(* IEC 61131-3 sources: Elmo_Master/Lasal_PRG/Elmo_EtherCAT_Test_4Axis/Class/SimulationSetup, 1 file *)

(* ---- SimulationSetup.st ---- *)
(*!
<Class
	Name               = "SimulationSetup"
	Revision           = "0.0"
	RealtimeTask       = "false"
	CyclicTask         = "false"
	BackgroundTask     = "false"
	Sigmatek           = "false"
	OSInterface        = "false"
	HighPriority       = "false"
	Automatic          = "false"
	UpdateMode         = "Prescan"
	SharedCommandTable = "true"
	Objectsize         = "(422,120)">
	<Channels>
		<Server Name="Axis_1" Visualized="false" Initialize="true" WriteProtected="false" Retentive="File"/>
		<Server Name="Axis_2" Visualized="false" Initialize="true" WriteProtected="false" Retentive="File"/>
		<Server Name="Axis_3" Visualized="false" Initialize="true" WriteProtected="false" Retentive="File"/>
		<Server Name="Axis_4" Visualized="false" Initialize="true" WriteProtected="false" Retentive="File"/>
		<Server Name="Axis_5" Visualized="false" Initialize="true" WriteProtected="false" Retentive="File"/>
		<Server Name="Axis_6" Visualized="false" Initialize="true" WriteProtected="false" Retentive="File"/>
		<Server Name="Axis_7" Visualized="false" Initialize="true" WriteProtected="false" Retentive="File"/>
		<Server Name="Axis_8" Visualized="false" Initialize="true" WriteProtected="false" Retentive="File"/>
		<Server Name="Axis_9" Visualized="false" Initialize="true" WriteProtected="false" Retentive="File"/>
		<Server Name="ClassSvr" Visualized="false" Initialize="false" WriteProtected="true" Retentive="false"/>
		<Client Name="Simul_Axis_1" Required="false" Internal="false"/>
		<Client Name="Simul_Axis_2" Required="false" Internal="false"/>
		<Client Name="Simul_Axis_3" Required="false" Internal="false"/>
		<Client Name="Simul_Axis_4" Required="false" Internal="false"/>
		<Client Name="Simul_Axis_5" Required="false" Internal="false"/>
		<Client Name="Simul_Axis_6" Required="false" Internal="false"/>
		<Client Name="Simul_Axis_7" Required="false" Internal="false"/>
		<Client Name="Simul_Axis_8" Required="false" Internal="false"/>
		<Client Name="Simul_Axis_9" Required="false" Internal="false"/>
	</Channels>
</Class>
*)
SimulationSetup : CLASS
  //Servers:
	ClassSvr 	: SvrChCmd_DINT;
	Axis_1 	: SvrCh_DINT;
	Axis_2 	: SvrCh_DINT;
	Axis_3 	: SvrCh_DINT;
	Axis_4 	: SvrCh_DINT;
	Axis_5 	: SvrCh_DINT;
	Axis_6 	: SvrCh_DINT;
	Axis_7 	: SvrCh_DINT;
	Axis_8 	: SvrCh_DINT;
	Axis_9 	: SvrCh_DINT;
  //Clients:
	Simul_Axis_1 	: CltCh_DINT;
	Simul_Axis_2 	: CltCh_DINT;
	Simul_Axis_3 	: CltCh_DINT;
	Simul_Axis_4 	: CltCh_DINT;
	Simul_Axis_5 	: CltCh_DINT;
	Simul_Axis_6 	: CltCh_DINT;
	Simul_Axis_7 	: CltCh_DINT;
	Simul_Axis_8 	: CltCh_DINT;
	Simul_Axis_9 	: CltCh_DINT;
  //Variables:
  //Functions:

	FUNCTION VIRTUAL GLOBAL Init;

	FUNCTION Write_Simul
		VAR_INPUT
			Index 	: DINT;
			Value 	: DINT;
		END_VAR;

	FUNCTION VIRTUAL GLOBAL Axis_1::Write
		VAR_INPUT
			input (EAX) 	: DINT;
		END_VAR
		VAR_OUTPUT
			result (EAX) 	: DINT;
		END_VAR;

	FUNCTION VIRTUAL GLOBAL Axis_2::Write
		VAR_INPUT
			input (EAX) 	: DINT;
		END_VAR
		VAR_OUTPUT
			result (EAX) 	: DINT;
		END_VAR;

	FUNCTION VIRTUAL GLOBAL Axis_3::Write
		VAR_INPUT
			input (EAX) 	: DINT;
		END_VAR
		VAR_OUTPUT
			result (EAX) 	: DINT;
		END_VAR;

	FUNCTION VIRTUAL GLOBAL Axis_4::Write
		VAR_INPUT
			input (EAX) 	: DINT;
		END_VAR
		VAR_OUTPUT
			result (EAX) 	: DINT;
		END_VAR;

	FUNCTION VIRTUAL GLOBAL Axis_5::Write
		VAR_INPUT
			input (EAX) 	: DINT;
		END_VAR
		VAR_OUTPUT
			result (EAX) 	: DINT;
		END_VAR;

	FUNCTION VIRTUAL GLOBAL Axis_6::Write
		VAR_INPUT
			input (EAX) 	: DINT;
		END_VAR
		VAR_OUTPUT
			result (EAX) 	: DINT;
		END_VAR;

	FUNCTION VIRTUAL GLOBAL Axis_7::Write
		VAR_INPUT
			input (EAX) 	: DINT;
		END_VAR
		VAR_OUTPUT
			result (EAX) 	: DINT;
		END_VAR;

	FUNCTION VIRTUAL GLOBAL Axis_8::Write
		VAR_INPUT
			input (EAX) 	: DINT;
		END_VAR
		VAR_OUTPUT
			result (EAX) 	: DINT;
		END_VAR;

	FUNCTION VIRTUAL GLOBAL Axis_9::Write
		VAR_INPUT
			input (EAX) 	: DINT;
		END_VAR
		VAR_OUTPUT
			result (EAX) 	: DINT;
		END_VAR;
  //Tables:
	FUNCTION @STD
		VAR_OUTPUT
			ret_code	: CONFSTATES;
		END_VAR;
	FUNCTION GLOBAL TAB @CT_;
END_CLASS;

FUNCTION VIRTUAL GLOBAL SimulationSetup::Init

  if _FirstScan = 1 then

    Write_Simul(Index:=1, Value:=Axis_1);
    Write_Simul(Index:=2, Value:=Axis_2);
    Write_Simul(Index:=3, Value:=Axis_3);
    Write_Simul(Index:=4, Value:=Axis_4);
    Write_Simul(Index:=5, Value:=Axis_5);
    Write_Simul(Index:=6, Value:=Axis_6);
    Write_Simul(Index:=7, Value:=Axis_7);
    Write_Simul(Index:=8, Value:=Axis_8);
    Write_Simul(Index:=9, Value:=Axis_9);

  end_if;

END_FUNCTION

FUNCTION VIRTUAL GLOBAL SimulationSetup::Axis_1::Write
	VAR_INPUT
		input (EAX) 	: DINT;
	END_VAR
	VAR_OUTPUT
		result (EAX) 	: DINT;
	END_VAR

	Axis_1 := input;
  Write_Simul(Index:=1, Value:=Axis_1);
	result := Axis_1;

END_FUNCTION

FUNCTION VIRTUAL GLOBAL SimulationSetup::Axis_2::Write
	VAR_INPUT
		input (EAX) 	: DINT;
	END_VAR
	VAR_OUTPUT
		result (EAX) 	: DINT;
	END_VAR

	Axis_2 := input;
  Write_Simul(Index:=2, Value:=Axis_2);
	result := Axis_2;

END_FUNCTION

FUNCTION VIRTUAL GLOBAL SimulationSetup::Axis_3::Write
	VAR_INPUT
		input (EAX) 	: DINT;
	END_VAR
	VAR_OUTPUT
		result (EAX) 	: DINT;
	END_VAR

	Axis_3 := input;
  Write_Simul(Index:=3, Value:=Axis_3);
	result := Axis_3;

END_FUNCTION

FUNCTION VIRTUAL GLOBAL SimulationSetup::Axis_4::Write
	VAR_INPUT
		input (EAX) 	: DINT;
	END_VAR
	VAR_OUTPUT
		result (EAX) 	: DINT;
	END_VAR

	Axis_4 := input;
  Write_Simul(Index:=4, Value:=Axis_4);
	result := Axis_4;

END_FUNCTION

FUNCTION VIRTUAL GLOBAL SimulationSetup::Axis_5::Write
	VAR_INPUT
		input (EAX) 	: DINT;
	END_VAR
	VAR_OUTPUT
		result (EAX) 	: DINT;
	END_VAR

	Axis_5 := input;
  Write_Simul(Index:=5, Value:=Axis_5);
	result := Axis_5;

END_FUNCTION

FUNCTION VIRTUAL GLOBAL SimulationSetup::Axis_6::Write
	VAR_INPUT
		input (EAX) 	: DINT;
	END_VAR
	VAR_OUTPUT
		result (EAX) 	: DINT;
	END_VAR

	Axis_6 := input;
  Write_Simul(Index:=6, Value:=Axis_6);
	result := Axis_6;

END_FUNCTION

FUNCTION VIRTUAL GLOBAL SimulationSetup::Axis_7::Write
	VAR_INPUT
		input (EAX) 	: DINT;
	END_VAR
	VAR_OUTPUT
		result (EAX) 	: DINT;
	END_VAR

	Axis_7 := input;
  Write_Simul(Index:=7, Value:=Axis_7);
	result := Axis_7;

END_FUNCTION

FUNCTION VIRTUAL GLOBAL SimulationSetup::Axis_8::Write
	VAR_INPUT
		input (EAX) 	: DINT;
	END_VAR
	VAR_OUTPUT
		result (EAX) 	: DINT;
	END_VAR

	Axis_8 := input;
  Write_Simul(Index:=8, Value:=Axis_8);
	result := Axis_8;

END_FUNCTION

FUNCTION VIRTUAL GLOBAL SimulationSetup::Axis_9::Write
	VAR_INPUT
		input (EAX) 	: DINT;
	END_VAR
	VAR_OUTPUT
		result (EAX) 	: DINT;
	END_VAR

	Axis_9 := input;
  Write_Simul(Index:=9, Value:=Axis_9);
	result := Axis_9;

END_FUNCTION

FUNCTION SimulationSetup::Write_Simul
	VAR_INPUT
		Index 	: DINT;
		Value 	: DINT;
	END_VAR

  case Index of

    1:
      Simul_Axis_1.Write(input:=Value);
    2:
      Simul_Axis_2.Write(input:=Value);
    3:
      Simul_Axis_3.Write(input:=Value);
    4:
      Simul_Axis_4.Write(input:=Value);
    5:
      Simul_Axis_5.Write(input:=Value);
    6:
      Simul_Axis_6.Write(input:=Value);
    7:
      Simul_Axis_7.Write(input:=Value);
    8:
      Simul_Axis_8.Write(input:=Value);
    9:
      Simul_Axis_9.Write(input:=Value);

  end_case;

END_FUNCTION
